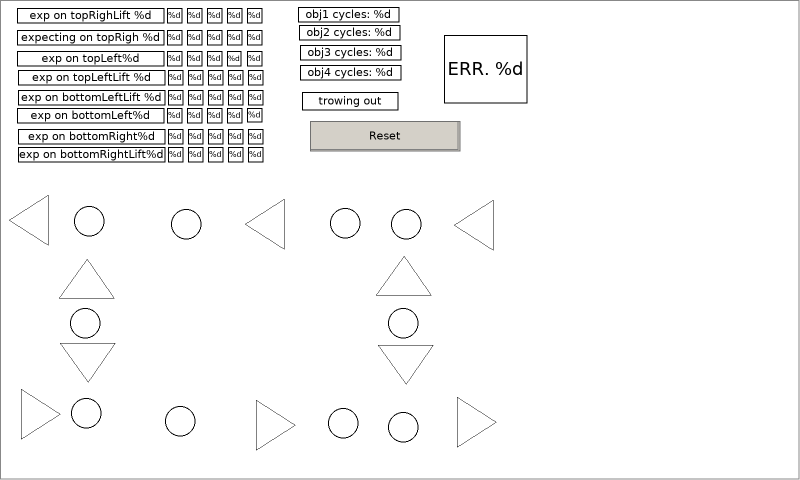
VISUALIZATION TouchScreen  // 800x480
    Rectangle (17,30 147x15), "expecting on topRigh %d", text variable: GVL.topRightExp
    Rectangle (167,30 15x15), "%d", text variable: GVL.topRightExpArr[1]
    Rectangle (187,30 15x15), "%d", text variable: GVL.topRightExpArr[2]
    Rectangle (207,30 15x15), "%d", text variable: GVL.topRightExpArr[3]
    Rectangle (227,30 15x15), "%d", text variable: GVL.topRightExpArr[4]
    Rectangle (247,30 15x15), "%d", text variable: GVL.topRightExpArr[5]
    Rectangle (17,8 147x15), "exp on topRighLift %d", text variable: GVL.topRightExp
    Rectangle (167,8 15x15), "%d", text variable: GVL.topRightLiftExpArr[1]
    Rectangle (187,8 15x15), "%d", text variable: GVL.topRightLiftExpArr[2]
    Rectangle (207,8 15x15), "%d", text variable: GVL.topRightLiftExpArr[3]
    Rectangle (227,8 15x15), "%d", text variable: GVL.topRightLiftExpArr[4]
    Rectangle (247,8 15x15), "%d", text variable: GVL.topRightLiftExpArr[5]
    Rectangle (17,51 147x15), "exp on topLeft%d", text variable: GVL.topRightExp
    Rectangle (167,51 15x15), "%d", text variable: GVL.topLeftExpArr[1]
    Rectangle (187,51 15x15), "%d", text variable: GVL.topLeftExpArr[2]
    Rectangle (207,51 15x15), "%d", text variable: GVL.topLeftExpArr[3]
    Rectangle (227,51 14x15), "%d", text variable: GVL.topLeftExpArr[4]
    Rectangle (247,51 15x15), "%d", text variable: GVL.topLeftExpArr[5]
    Rectangle (18,70 147x15), "exp on topLeftLift %d", text variable: GVL.topRightExp
    Rectangle (168,70 15x15), "%d", text variable: GVL.topLeftLiftExpArr[1]
    Rectangle (188,70 15x15), "%d", text variable: GVL.topLeftLiftExpArr[2]
    Rectangle (208,70 15x15), "%d", text variable: GVL.topLeftLiftExpArr[3]
    Rectangle (228,70 15x15), "%d", text variable: GVL.topLeftLiftExpArr[4]
    Rectangle (248,70 15x15), "%d", text variable: GVL.topLeftLiftExpArr[5]
    Rectangle (18,90 147x15), "exp on bottomLeftLift %d", text variable: GVL.topRightExp
    Rectangle (168,90 15x15), "%d", text variable: GVL.bottomLeftLiftExpArr[1]
    Rectangle (188,90 15x15), "%d", text variable: GVL.bottomLeftLiftExpArr[2]
    Rectangle (208,90 15x15), "%d", text variable: GVL.bottomLeftLiftExpArr[3]
    Rectangle (228,90 15x15), "%d", text variable: GVL.bottomLeftLiftExpArr[4]
    Rectangle (248,90 15x15), "%d", text variable: GVL.bottomLeftLiftExpArr[5]
    Rectangle (17,108 147x15), "exp on bottomLeft%d", text variable: GVL.topRightExp
    Rectangle (167,108 15x15), "%d", text variable: GVL.bottomLeftExpArr[1]
    Rectangle (187,108 15x15), "%d", text variable: GVL.bottomLeftExpArr[2]
    Rectangle (207,108 15x15), "%d", text variable: GVL.bottomLeftExpArr[3]
    Rectangle (227,108 15x15), "%d", text variable: GVL.bottomLeftExpArr[4]
    Rectangle (247,108 15x14), "%d", text variable: GVL.bottomLeftExpArr[5]
    Rectangle (18,129 147x15), "exp on bottomRight%d", text variable: GVL.topRightExp
    Rectangle (168,129 15x15), "%d", text variable: GVL.bottomRightExpArr[1]
    Rectangle (188,129 15x15), "%d", text variable: GVL.bottomRightExpArr[2]
    Rectangle (208,129 15x15), "%d", text variable: GVL.bottomRightExpArr[3]
    Rectangle (228,129 15x15), "%d", text variable: GVL.bottomRightExpArr[4]
    Rectangle (248,129 15x15), "%d", text variable: GVL.bottomRightExpArr[5]
    Rectangle (18,147 147x15), "exp on bottomRightLift%d", text variable: GVL.topRightExp
    Rectangle (168,147 15x15), "%d", text variable: GVL.bottomRightLiftExpArr[1]
    Rectangle (188,147 15x15), "%d", text variable: GVL.bottomRightLiftExpArr[2]
    Rectangle (208,147 15x15), "%d", text variable: GVL.bottomRightLiftExpArr[3]
    Rectangle (228,147 15x15), "%d", text variable: GVL.bottomRightLiftExpArr[4]
    Rectangle (248,147 15x15), "%d", text variable: GVL.bottomRightLiftExpArr[5]
    Rectangle (299,25 101x15), "obj2 cycles: %d", text variable: GVL.obj2
    Rectangle (298,7 101x15), "obj1 cycles: %d", text variable: GVL.obj1
    Rectangle (300,45 101x15), "obj3 cycles: %d", text variable: GVL.obj3
    Rectangle (300,65 101x15), "obj4 cycles: %d", text variable: GVL.obj4
    Rectangle (302,92 96x18), "trowing out", colour toggle: GVL.trowingObjectOut
    Ellipse (388,308 30x30), colour toggle: GVL.rightLiftOptical_IB
    Ellipse (330,208 30x30), colour toggle: GVL.topRight_IB
    Ellipse (171,209 30x30), colour toggle: GVL.topLeft_IB
    Ellipse (74,206 30x30), colour toggle: GVL.leftLiftUpPosition_IB
    Ellipse (391,209 30x30), colour toggle: GVL.rightLiftUpPosition_IB
    Ellipse (388,412 30x30), colour toggle: GVL.rightLiftDownPosition_IB
    Ellipse (328,408 30x30), colour toggle: GVL.bottomRight_IB
    Ellipse (165,406 30x30), colour toggle: GVL.bottomLeft_IB
    Ellipse (71,398 30x30), colour toggle: GVL.leftLiftDownPosition_IB
    Ellipse (70,308 30x30), colour toggle: GVL.leftLiftOptical_IB
    Polygon (9,220) (48,195) (48,220) (48,230) (48,245), colour toggle: GVL.leftLiftBeltLeft_OB
        OnMouseDown: toggle GVL.leftLiftBeltLeft_OB
    Polygon (245,224) (284,199) (284,224) (284,234) (284,249), colour toggle: GVL.topBeltLeft_OB
        OnMouseDown: toggle GVL.topBeltLeft_OB
    Polygon (454,225) (493,200) (493,225) (493,235) (493,250), colour toggle: GVL.rightLiftBeltLeft_OB
        OnMouseDown: toggle GVL.rightLiftBeltLeft_OB
    Polygon (60,414) (21,389) (21,414) (21,424) (21,439), colour toggle: GVL.leftLiftBeltRight_OB
        OnMouseDown: toggle GVL.leftLiftBeltRight_OB
    Polygon (295,425) (256,400) (256,425) (256,435) (256,450), colour toggle: GVL.bottomBeltRight_OB
        OnMouseDown: toggle GVL.bottomBeltRight_OB
    Polygon (496,422) (457,397) (457,422) (457,432) (457,447), colour toggle: GVL.rightLiftBeltRight_OB
        OnMouseDown: toggle GVL.rightLiftBeltRight_OB
    Polygon (88,382) (60,343) (88,343) (100,343) (115,343), colour toggle: GVL.leftLiftDown_OB
        OnMouseDown: toggle GVL.leftLiftUp_OB
    Polygon (406,384) (378,345) (406,345) (418,345) (433,345), colour toggle: GVL.rightLiftDown_OB
        OnMouseDown: toggle GVL.rightLiftDown_OB
    Polygon (404,256) (376,295) (404,295) (416,295) (431,295), colour toggle: GVL.rightLiftUp_OB
        OnMouseDown: toggle GVL.rightLiftUp_OB
    Polygon (87,259) (59,298) (87,298) (99,298) (114,298), colour toggle: GVL.leftLiftUp_OB
        OnMouseDown: toggle GVL.leftLiftUp_OB
    Button (310,121 150x30), "Reset"
        OnMouseDown: toggle resetAll
        OnMouseUp: toggle resetAll
    Rectangle (444,35 83x68), "ERR. %d", text variable: ERR
END_VISUALIZATION

(* stored: Version 1.1.0.1, ProductVersion 3.1.4018.5
   Visu TouchScreen: Id {b71f7a52-4e29-458a-b222-0c731d3d5203} *)
